{attribute 'linkalways'} 
{attribute 'no_explicit_call' := 'This FB is a CLASS and must be accessed using methods or properties'}
{attribute 'enable_dynamic_creation'}
FUNCTION_BLOCK FINAL GT_WORD EXTENDS Node
VAR
	in1 : _WORD(0);
	in2 : _WORD(0);
	out : _BOOL(FALSE);
END_VAR

METHOD PUBLIC Clone : I_Node
VAR
	pNode : POINTER TO GT_WORD;
END_VAR
pNode := __NEW(GT_WORD);
Clone := pNode^;
END_METHOD

METHOD FB_init : BOOL
VAR_INPUT
	bInitRetains : BOOL; // if TRUE, the retain variables are initialized (warm start / cold start)
	bInCopyCode : BOOL;  // if TRUE, the instance afterwards gets moved into the copy code (online change)
END_VAR
AddInput('in1',THIS^.in1);
AddInput('in2',THIS^.in2);
AddOutput('out', THIS^.out);
END_METHOD

METHOD PROTECTED OnExecute
VAR
END_VAR
out.Value := in1.Value > in2.Value;
END_METHOD

END_FUNCTION_BLOCK

(* stored: Version 1.1.0.1, ProductVersion 3.1.4024.15
   POU GT_WORD: Id {1bd976d3-629c-4ccf-8cca-3b46f46203bf}, SpecialFunc None
   Folder Constructor: Id {f7deb9c8-8341-4e94-8a0d-d0bfc5893449}
   Method Clone: Id {6022c46b-5631-4e73-94eb-de94c12a8769}
   Method FB_init: Id {baffff07-3e4b-4471-8344-0882e47ccf26}
   Method OnExecute: Id {14e34f91-51a2-4190-8032-ac44443bdd28} *)
